PROGRAM P1_02_Batch
VAR
		fbBatch					:FB_Batch;
		fbBatchLog				:FB_BatchLog;
END_VAR
VAR PERSISTENT
	tonBatchTime				:FB_TONP;
END_VAR
VAR // added by the converter: edge detectors and wires of the graphical bodies
    _rt1, _rt2, _rt3, _rt4, _rt5, _rt6, _rt7, _rt8, _rt9, _rt10 : R_TRIG;
    _w1, _w2 : BOOL;
END_VAR

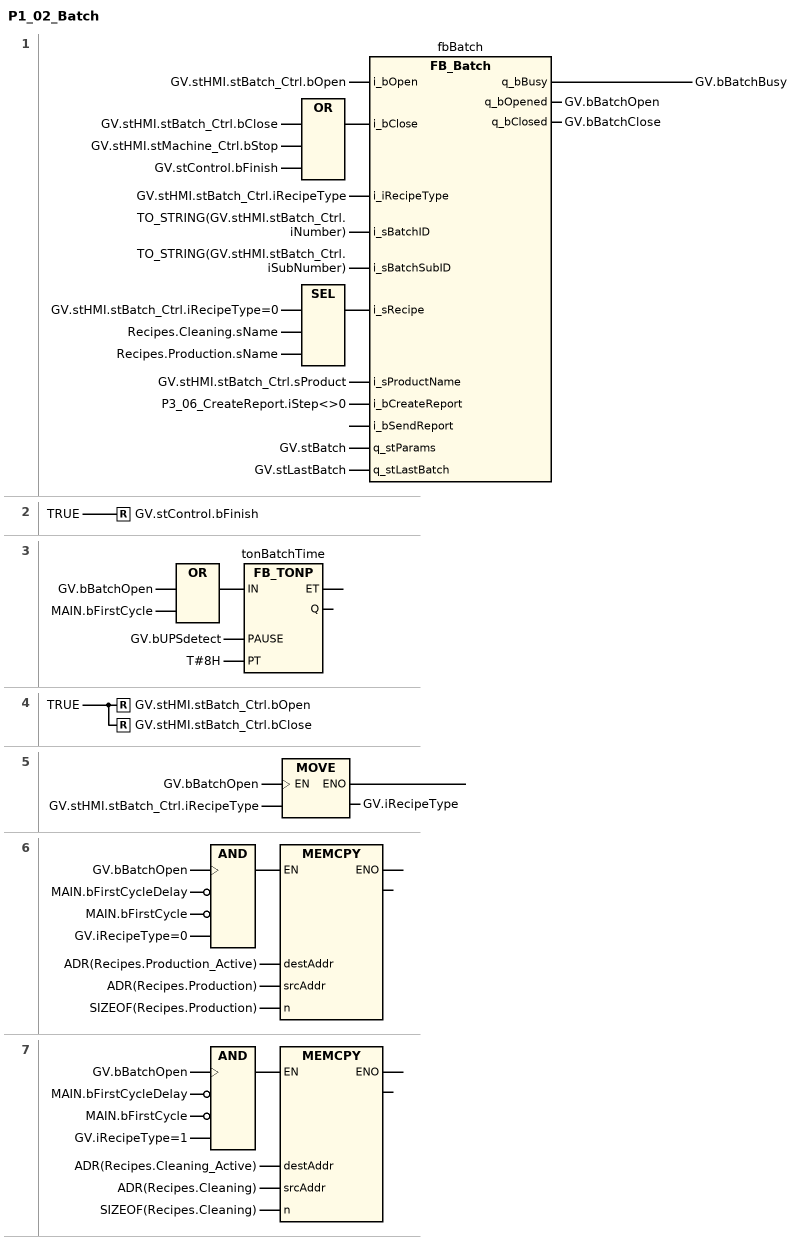
// NETWORK 1
fbBatch(
    i_bOpen := GV.stHMI.stBatch_Ctrl.bOpen,
    i_bClose := GV.stHMI.stBatch_Ctrl.bClose OR GV.stHMI.stMachine_Ctrl.bStop OR GV.stControl.bFinish,
    i_iRecipeType := GV.stHMI.stBatch_Ctrl.iRecipeType,
    i_sBatchID := TO_STRING(GV.stHMI.stBatch_Ctrl.iNumber),
    i_sBatchSubID := TO_STRING(GV.stHMI.stBatch_Ctrl.iSubNumber),
    i_sRecipe := SEL(GV.stHMI.stBatch_Ctrl.iRecipeType=0, Recipes.Cleaning.sName, Recipes.Production.sName),
    i_sProductName := GV.stHMI.stBatch_Ctrl.sProduct,
    i_bCreateReport := P3_06_CreateReport.iStep<>0,
    q_stParams := GV.stBatch,
    q_stLastBatch := GV.stLastBatch,
    q_bOpened => GV.bBatchOpen,
    q_bClosed => GV.bBatchClose); // FB_Batch
GV.bBatchBusy := fbBatch.q_bBusy;

// NETWORK 2
GV.stControl.bFinish R= TRUE;

// NETWORK 3
tonBatchTime(IN := GV.bBatchOpen OR MAIN.bFirstCycle, PAUSE := GV.bUPSdetect, PT := T#8H); // FB_TONP

// NETWORK 4
GV.stHMI.stBatch_Ctrl.bOpen R= TRUE;
GV.stHMI.stBatch_Ctrl.bClose R= TRUE;

// NETWORK 5
_rt1(CLK := GV.bBatchOpen);
IF _rt1.Q THEN GV.iRecipeType := GV.stHMI.stBatch_Ctrl.iRecipeType; END_IF

// NETWORK 6
_rt2(CLK := GV.bBatchOpen);
IF _rt2.Q AND NOT MAIN.bFirstCycleDelay AND NOT MAIN.bFirstCycle AND (GV.iRecipeType=0) THEN
    MEMCPY(destAddr := ADR(Recipes.Production_Active), srcAddr := ADR(Recipes.Production), n := SIZEOF(Recipes.Production));
END_IF

// NETWORK 7
_rt3(CLK := GV.bBatchOpen);
IF _rt3.Q AND NOT MAIN.bFirstCycleDelay AND NOT MAIN.bFirstCycle AND (GV.iRecipeType=1) THEN
    MEMCPY(destAddr := ADR(Recipes.Cleaning_Active), srcAddr := ADR(Recipes.Cleaning), n := SIZEOF(Recipes.Cleaning));
END_IF

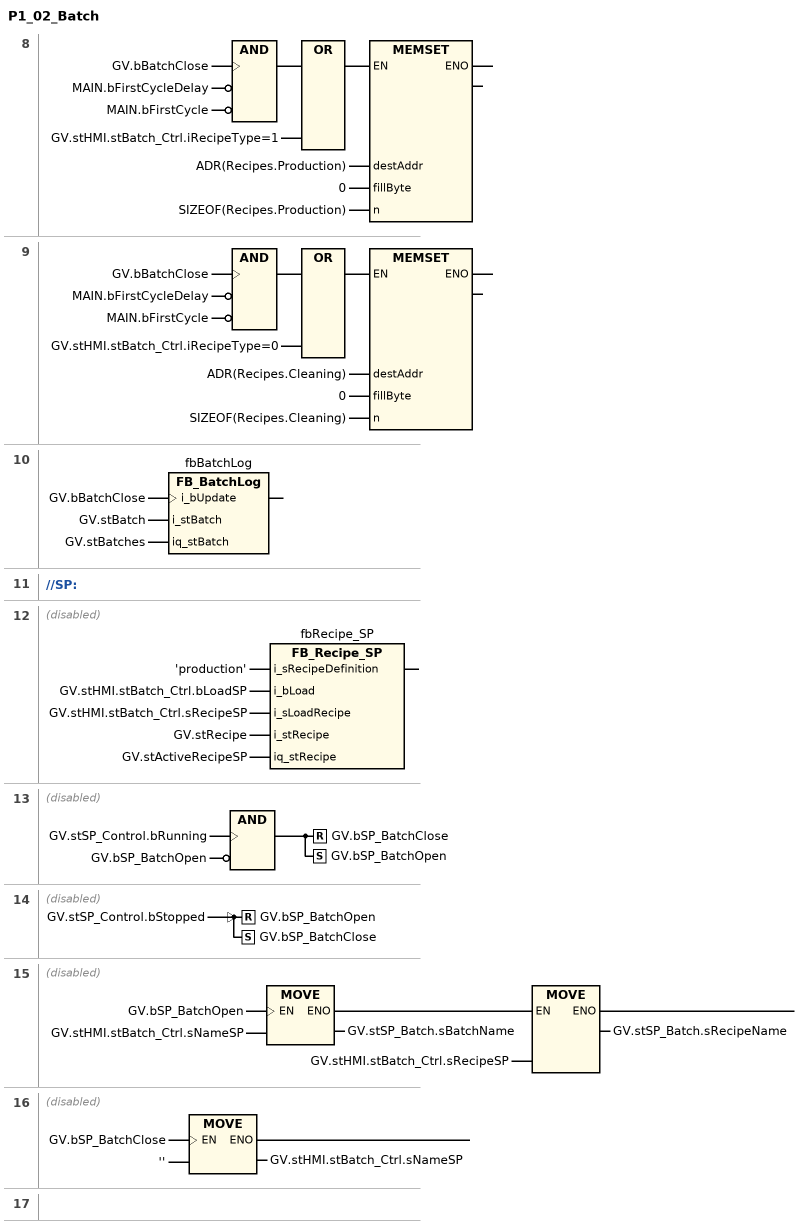
// NETWORK 8
_rt4(CLK := GV.bBatchClose);
IF _rt4.Q AND NOT MAIN.bFirstCycleDelay AND NOT MAIN.bFirstCycle OR (GV.stHMI.stBatch_Ctrl.iRecipeType=1) THEN
    MEMSET(destAddr := ADR(Recipes.Production), fillByte := 0, n := SIZEOF(Recipes.Production));
END_IF

// NETWORK 9
_rt5(CLK := GV.bBatchClose);
IF _rt5.Q AND NOT MAIN.bFirstCycleDelay AND NOT MAIN.bFirstCycle OR (GV.stHMI.stBatch_Ctrl.iRecipeType=0) THEN
    MEMSET(destAddr := ADR(Recipes.Cleaning), fillByte := 0, n := SIZEOF(Recipes.Cleaning));
END_IF

// NETWORK 10
_rt6(CLK := GV.bBatchClose);
fbBatchLog(i_bUpdate := _rt6.Q, i_stBatch := GV.stBatch, iq_stBatch := GV.stBatches); // FB_BatchLog

// NETWORK 11
// label: //SP

// NETWORK 12 (disabled)
// fbRecipe_SP(
//     i_sRecipeDefinition := 'production',
//     i_bLoad := GV.stHMI.stBatch_Ctrl.bLoadSP,
//     i_sLoadRecipe := GV.stHMI.stBatch_Ctrl.sRecipeSP,
//     i_stRecipe := GV.stRecipe,
//     iq_stRecipe := GV.stActiveRecipeSP); // FB_Recipe_SP

// NETWORK 13 (disabled)
// _rt7(CLK := GV.stSP_Control.bRunning);
// _w1 := _rt7.Q AND NOT GV.bSP_BatchOpen;
// GV.bSP_BatchClose R= _w1;
// GV.bSP_BatchOpen S= _w1;

// NETWORK 14 (disabled)
// _rt8(CLK := GV.stSP_Control.bStopped);
// GV.bSP_BatchOpen R= _rt8.Q;
// GV.bSP_BatchClose S= _rt8.Q;

// NETWORK 15 (disabled)
// _rt9(CLK := GV.bSP_BatchOpen);
// _w2 := _rt9.Q;
// IF _w2 THEN GV.stSP_Batch.sBatchName := GV.stHMI.stBatch_Ctrl.sNameSP; END_IF
// IF _w2 THEN GV.stSP_Batch.sRecipeName := GV.stHMI.stBatch_Ctrl.sRecipeSP; END_IF

// NETWORK 16 (disabled)
// _rt10(CLK := GV.bSP_BatchClose);
// IF _rt10.Q THEN GV.stHMI.stBatch_Ctrl.sNameSP := ''; END_IF

// NETWORK 17

END_PROGRAM

(* stored: Version 1.1.0.1, ProductVersion 3.1.4026.13
   POU P1_02_Batch: Id {fde4e061-7102-4637-ad9f-2ce99741e8b7}, SpecialFunc None *)
